Staubli VAL3: PCData.dtx

mdesc mNomSpeed
public frame fFrame = {fatherId=world[0]}
public num nNum[2]
public pointRx pPos[2]
  [0] = {fatherId=world[0]}
  [1] = {fatherId=world[0]}
public string sString
public trsf trTrsf[2]
public tool tTool[2]
  [0] = {fatherId=flange[0], ioLink=valve1}
  [1] = {fatherId=flange[0], ioLink=valve1}
public jointRx jJ[2]
public bool bBool
